// Some of the bits are 
FUNCTION F_GetKL306xState
VAR_INPUT
	KL306xState : stKL306x_ChannelStatus;
END_VAR
VAR_OUTPUT
	Underrange : BOOL;
	Overrange : BOOL;
	ProcessData_EQ_Limit1 : BOOL;
	ProcessData_GT_Limit1 : BOOL;
	ProcessData_LT_Limit1 : BOOL;
	Limit1NotEnabled : BOOL;
	ProcessData_EQ_Limit2 : BOOL;
	ProcessData_GT_Limit2 : BOOL;
	ProcessData_LT_Limit2 : BOOL;
	Limit2NotEnabled : BOOL;
	Error : BOOL;
END_VAR

Underrange := KL306xState.Underrange;
Overrange := KL306xState.Overrange;

ProcessData_EQ_Limit1 := KL306xState.Limit1Bit_1 AND KL306xState.Limit1Bit_0;
ProcessData_GT_Limit1 := KL306xState.Limit1Bit_1 AND NOT KL306xState.Limit1Bit_0;
ProcessData_LT_Limit1 := NOT KL306xState.Limit1Bit_1 AND KL306xState.Limit1Bit_0;
Limit1NotEnabled := NOT KL306xState.Limit1Bit_1 AND NOT KL306xState.Limit1Bit_0;

ProcessData_EQ_Limit2 := KL306xState.Limit2Bit_1 AND KL306xState.Limit2Bit_0;
ProcessData_GT_Limit2 := KL306xState.Limit2Bit_1 AND NOT KL306xState.Limit2Bit_0;
ProcessData_LT_Limit2 := NOT KL306xState.Limit2Bit_1 AND KL306xState.Limit2Bit_0;
Limit2NotEnabled := NOT KL306xState.Limit2Bit_1 AND NOT KL306xState.Limit2Bit_0;

Error := KL306xState.Error;

END_FUNCTION

(* stored: Version 1.1.0.1, ProductVersion 3.1.4024.9
   POU F_GetKL306xState: Id {fed3897d-ed45-462c-815a-c32436a369f0}, SpecialFunc None *)
